Fanuc KAREL source: compact_preamble.KL

PROGRAM KT00150
%NOLOCKGROUP
VAR
Y1 : ARRAY[2] OF BYTE
Y2 : ARRAY[2] OF BYTE
OUT:REAL
BEGIN
Y1[1]=2
Y2[1]=3
Y1[1]=2
Y2[1]=3
OUT=((Y1[1] DIV Y2[1]))
END KT00150
